{attribute 'qualified_only'}
VAR_GLOBAL
	fbHMIControl	: FB_HMIControl ; // HMI control function
	nStartVisu		: E_BaseVisu := E_BaseVisu.Idle ;
	nSelectedMessage : INT; 
END_VAR

(* stored: Version 1.1.0.1, ProductVersion 3.1.4024.5
   GVL GVL_HMI: Id {fb24c9f0-ea70-489c-b3f0-65a490c6fceb} *)
